(* IEC 61131-3 sources: CodesysTest/export/SX_1195.dev/Plc Logic/Application/PRJ Specific/Motion/Motors/Oriental AZD/AZD4A-KED/FB_AZDKABase.pou, 4 files *)

(* ---- FB_AZDKABase.pou.st ---- *)
(*#-#-#-#-#-#-#-#-#-#---Declaration---#-#-#-#-#-#-#-#-#-#-#-#-#*)

FUNCTION_BLOCK FB_AZDKABase EXTENDS Axis_REF
VAR_INPUT
	jogForwardCMD : BOOL;
	jogReverseCMD : BOOL;
	iErrorCode : UINT;
	iModeOfOperation : SINT;
	iStatusword : UINT;
	iActualVelocity : DINT;
	iActualPosition : DINT;
END_VAR
VAR_OUTPUT
	oControlword : UINT;
	oModeOfOperation : eAZDProfileMode;
	oTargetPosition : DINT;
	oProfileVelocity : UDINT;
	oProfileAcceleration : UDINT;
	oProfileDeceleration : UDINT;
	oProfilePushCurrent : INT;
	oProfileOperationalCurrent : INT;
	alarmCode : eOrientalAZDriveFaults;
	actualPositonInInches : REAL;
END_VAR
VAR
	_resetONS : FB_ONS;
	_jogForwardONS : FB_ONS;
	_jogReverseONS : FB_ONS;
	_relativeONS : FB_ONS;
	_zHomeONS : FB_ONS;
	_absoluteONS : FB_ONS;
	_absoluteTorqueONS : FB_ONS;
	_homeONS : FB_ONS;
	_errorONS : FB_ONS;
	_haltONS : Standard.R_TRIG;
	_statusword : FB_AZDStatus;
	_controlword : FB_AZDControl;
	_state : eAxisREFMotionState;
	_startupState : eAZDPowerupState;
	_motorExcitationDelayTimer : Standard.TON := (PT := T#250MS);
	_resetSignalPulseTON : Standard.TON := (PT := T#50MS);
	_codetemp : DWORD;
END_VAR
(*#-#-#-#-#-#-#-#-#-#---Implementation---#-#-#-#-#-#-#-#-#-#-#-#-#*)

//
//  FB_AZDOrientalMotor
//  FB/FB_AZDOrientalMotor
//
//  Created by Evan Ische on 6/13/2022.
//  Copyright (C) 2022 Sharp Packaging Systems By Pregis. All rights reserved.
//

//
operational := EnableAxisOps();

//
_resetSignalPulseTON.IN := ackError;
_controlword.FaultReset := _statusword.fault AND ackError AND NOT _resetSignalPulseTON.Q;

//diagnostic code - delete me
IF _statusword.fault AND ackError AND NOT _resetSignalPulseTON.Q THEN
	_codetemp := _codetemp;
END_IF

// Status bits read from the AZD4A drive
_statusword(
	mode := modeOfOperation,
	data := iStatusword);

// Control bits written to the AZD4A drive
_controlword(
	mode := modeOfOperation,
	data => oControlword
);

// Active Alarm
alarmCode := OSCAT_BASIC.BYTE_OF_DWORD(iErrorCode,0);
isHomed := _statusword.homingAttained;
IF alarmCode <> 0 THEN
	_codetemp := alarmCode;
END_IF
_errorONS(CLK := _statusword.fault);

error := _statusword.fault;
// IF _errorONS.OSR THEN
// 	error := TRUE;
// END_IF
// Convert Distance setpoint to steps.  Reverse polarity for display purposes if needed.
actualPositonInInches := (actPos / TO_REAL(axisData.config.stepsPerInch));
IF axisData.config.reversePolarity THEN
    actualPositonInInches := actualPositonInInches * -1;
END_IF

// Perform move on rising edge
_haltONS(CLK := Halt);
_relativeONS(CLK := MoveRel);
_absoluteONS(CLK := MoveAbs);
_absoluteTorqueONS(CLK := moveAbsTorque);
_homeONS(CLK := startHoming);
IF _homeONS.OSR THEN
	_controlword.HomingOperationStart:=TRUE;
END_IF
// Write data from drive to local variables
actPos := TO_REAL(iActualPosition) + zeroOffset * axisData.config.stepsPerInch;
actVel := TO_REAL(iActualVelocity);

// Write data to drive from local variables
oTargetPosition := TO_DINT(TargetPositionInSteps);
oProfileVelocity := TO_UDINT(ProfileVelocityInEngUnits);
oProfileAcceleration := TO_UDINT(EngUnitsToHz(ProfileAcceleration));
oProfileDeceleration := TO_UDINT(EngUnitsToHz(ProfileDeceleration));
oProfilePushCurrent := TO_INT(profilePushCurrentLimit * 10.0);
IF push THEN
	oProfileOperationalCurrent := TO_INT(defaultCurrent * 10.0);
ELSE
	oProfileOperationalCurrent := TO_INT(profileCurrentLimit * 10.0);
END_IF

oModeOfOperation := modeOfOperation;

// On rising edge start moving, on falling edge halt
_jogForwardONS(CLK := jogForwardCMD);
_jogReverseONS(CLK := jogReverseCMD);
IF _jogForwardONS.OSR OR _jogReverseONS.OSR THEN
	CASE axisData.jogType OF
		eDiscreteMotionType.Relative:
			profileAcceleration := axisData.jogProfile.acceleration;
			profileDeceleration := axisData.jogProfile.deceleration;
			profileVelocity := axisData.jogProfile.velocity;
			targetPosDist := axisData.jogProfile.position;
			IF _jogReverseONS.OSR THEN
				targetPosDist := targetPosDist * -1;
			END_IF
		eDiscreteMotionType.Absolute:
			profileAcceleration := axisData.jogProfile.acceleration;
			profileDeceleration := axisData.jogProfile.deceleration;
			profileVelocity := axisData.jogProfile.velocity;
			targetPosDist := axisData.jogProfile.maxPosition;
			IF _jogReverseONS.OSR THEN
				targetPosDist := axisData.jogProfile.minPosition;
			END_IF
	END_CASE
	_state := eAxisREFMotionState.Jog;
ELSIF _jogForwardONS.OSF OR _jogReverseONS.OSF OR _haltONS.Q THEN
	_state := eAxisREFMotionState.Halt;
END_IF

(* ---- EnableAxisOps.m.st ---- *)
(*#-#-#-#-#-#-#-#-#-#---Declaration---#-#-#-#-#-#-#-#-#-#-#-#-#*)

METHOD PRIVATE EnableAxisOps : BOOL
VAR_INPUT
END_VAR
VAR
	_driveEnabledONS : FB_ONS;
END_VAR(*#-#-#-#-#-#-#-#-#-#---Implementation---#-#-#-#-#-#-#-#-#-#-#-#-#*)

// 250MS wait period from when the status operational bit goes high, until a command can be processed.
_motorExcitationDelayTimer();
_motorExcitationDelayTimer.IN := _startupState = eAZDPowerupState.Operational;
EnableAxisOps := _motorExcitationDelayTimer.Q;

// If E-Stopped, or Comm Failure clear state machine
IF NOT driveEnable OR operational AND (NOT _statusword.voltageEnabled OR NOT _statusword.switchedOn) THEN
	_startupState := eAZDPowerupState.Idle;
END_IF
_driveEnabledONS(CLK := driveEnable);

// Startup state machine
CASE _startupState OF
	eAZDPowerupState.Idle:
		_controlword.Clear();
		IF _statusword.switchOnDisabled THEN
			IF driveEnable THEN
				_startupState := eAZDPowerupState.Shutdown; // Doesnt mean shutdown
			END_IF
// 		ELSIF _driveEnabledONS.OSR AND _statusword.readyToSwitchOn AND NOT _statusword.switchedOn AND NOT _statusword.operationEnabled  THEN
// 			_startupState := eAZDPowerupState.Shutdown; // Doesnt mean shutdown
		END_IF

	eAZDPowerupState.Shutdown:
		_controlword.Shutdown();
		IF _statusword.readyToSwitchOn  THEN
			_startupState := eAZDPowerupState.SwitchOn;
		END_IF

	eAZDPowerupState.SwitchOn:
		_controlword.SwitchOn();
		IF _statusword.switchedOn THEN
			_startupState := eAZDPowerupState.SwitchOnEnableOp;
		END_IF

	eAZDPowerupState.SwitchOnEnableOp:
		_controlword.SwitchOnEnableOp();
		IF _statusword.operationEnabled THEN
			_startupState := eAZDPowerupState.Operational;
		END_IF

END_CASE

(* ---- EngUnitsToHz.m.st ---- *)
(*#-#-#-#-#-#-#-#-#-#---Declaration---#-#-#-#-#-#-#-#-#-#-#-#-#*)

METHOD EngUnitsToHz : REAL
VAR_INPUT
	engineeringUnits : REAL;
END_VAR
(*#-#-#-#-#-#-#-#-#-#---Implementation---#-#-#-#-#-#-#-#-#-#-#-#-#*)

EngUnitsToHz := ((engineeringUnits * axisData.config.rotationsPerInch) * 10000);

(* ---- GetPositionInInches.m.st ---- *)
(*#-#-#-#-#-#-#-#-#-#---Declaration---#-#-#-#-#-#-#-#-#-#-#-#-#*)

METHOD PRIVATE GetPositionInInches : BOOL
VAR_INPUT
END_VAR
(*#-#-#-#-#-#-#-#-#-#---Implementation---#-#-#-#-#-#-#-#-#-#-#-#-#*)
